Universal Robots PolyScope program: center_object_5cm_open.urp

Program center_object_5cm_open (installation=default directory=/programs/wrs2020 createdIn=5.7.0.90932 lastSavedIn=5.9.1.1031110 robotSerialNumber=20205500180)
Calibrated DH parameters: a=[0, -0.425, -0.3922, 0, 0, 0]; d=[0.1625, 0, 0, 0.1333, 0.0997, 0.0996]; alpha=[1.570796, 0, 0, 1.570796, -1.570796, 0]; deltaTheta=[0, 0, 0, 0, 0, 0]
Robot Program (runOnlyOnce=true)
  URCap Gripper (Robotiq_Grippers, Robotiq Inc.) dataModel(position=100.0, force=0.0, speed=0.0, positionInDouble=100.0, forceInDouble=0.0, speedInDouble=0.0, slaveIds=[9], blocking=true)
  URCap Gripper (Robotiq_Grippers, Robotiq Inc.) dataModel(position=56.470588235294116, force=100.0, speed=0.0, positionInDouble=56.470588235294116, forceInDouble=100.0, speedInDouble=0.0, slaveIds=[9], blocking=true)
  MoveJ speed 180 deg/s, acceleration 800 deg/s^2 (useActiveTCP=true) feature=Base
    Waypoint turn_right (Relative): relativeFromPosition TCP in base x=218.277 y=-500.897 z=48.153 mm, rx=-2.1842 ry=2.228 rz=-0.024 rad; joints [98.784, -72.216, 112.616, -130.369, -88.16, -80.001] deg; TCP offset x=0 y=0 z=165 mm, rx=0 ry=0 rz=0 rad; TCP in base x=218.316 y=-500.86 z=48.143 mm, rx=0.031 ry=3.1153 rz=0.0068 rad; joints [98.786, -72.217, 112.618, -130.367, -88.154, 10.001] deg
  URCap Gripper (Robotiq_Grippers, Robotiq Inc.) dataModel(position=100.0, force=0.0, speed=0.0, positionInDouble=100.0, forceInDouble=0.0, speedInDouble=0.0, slaveIds=[9], blocking=true)
  URCap Gripper (Robotiq_Grippers, Robotiq Inc.) dataModel(position=56.470588235294116, force=100.0, speed=0.0, positionInDouble=56.470588235294116, forceInDouble=100.0, speedInDouble=0.0, slaveIds=[9], blocking=true)
  MoveJ speed 180 deg/s, acceleration 1000 deg/s^2 (useActiveTCP=true) feature=Base
    Waypoint turn_left (Relative): relativeFromPosition TCP in base x=218.287 y=-500.864 z=48.112 mm, rx=0.031 ry=3.1154 rz=0.0069 rad; joints [98.785, -72.214, 112.618, -130.367, -88.158, 9.999] deg; TCP in base x=218.294 y=-500.846 z=48.105 mm, rx=-2.1841 ry=2.228 rz=-0.0238 rad; joints [98.786, -72.214, 112.619, -130.366, -88.158, -79.999] deg
  URCap Gripper (Robotiq_Grippers, Robotiq Inc.) dataModel(position=100.0, force=0.0, speed=0.0, positionInDouble=100.0, forceInDouble=0.0, speedInDouble=0.0, slaveIds=[9], blocking=true)
  URCap Gripper (Robotiq_Grippers, Robotiq Inc.) dataModel(position=56.470588235294116, force=100.0, speed=0.0, positionInDouble=56.470588235294116, forceInDouble=100.0, speedInDouble=0.0, slaveIds=[9], blocking=true)
